// Device/Application/workflowCore
PROGRAM workflowCore
VAR 
	right2All:BOOL;//右扫切全扫标志
	left2All:BOOL;//左扫切全扫标志
	all2Right:BOOL;//全扫切右扫标志
	all2Left:BOOL;//全扫切左扫标志
	leftSweeperSwingOutTemp:BOOL;//左扫摆出中间变量
	rightSweeperSwingOutTemp:BOOL;//右扫摆出中间变量
	ton1:TON;//左扫盘延时下放定时器
	ton2:TON;//左扫盘下放控制延时定时器
	ton3:TON;//右扫盘延时下放定时器
	ton4:TON;//右扫盘下放控制延时定时器
	ton5:TON;//吸嘴延时下降定时器
	ton6:TON;//吸嘴下降持续时间定时器
	ton7:TON;//左扫延时旋转定时器
	ton8:TON;//右扫延时旋转定时器
	ton9:TON;//全扫延时旋转定时器
	ton10:TON;//右扫切全扫定时器
	ton11:TON;//左扫切全扫定时器
	ton12:TON;//全扫切右扫定时器
	ton13:TON;//全扫切左扫定时器
	ton14:TON;//左扫盘上升定时器
	ton15:TON;//右扫盘上升定时器
	ton16:TON;//吸嘴上升定时器
	ton17:TON;//中喷杆球阀定时器
	ton18:TON;//左喷杆球阀定时器
	ton19:TON;//右喷杆球阀定时器
	ton20:TON;//喷雾降尘泵定时器
	tof1:TOF;//左扫盘延时回收定时器
	tof2:TOF;//右扫盘延时回收定时器
	rTrigger1:R_TRIG;//全洗扫上升沿触发
	rTrigger2:R_TRIG;//左洗扫上升沿触发
	rTrigger3:R_TRIG;//右洗扫上升沿触发
	rTrigger4:R_TRIG;//全扫路上升沿触发
	rTrigger5:R_TRIG;//左扫路上升沿触发
	rTrigger6:R_TRIG;//右扫路上升沿触发
	rTrigger7:R_TRIG;//系统工作状态上升沿触发
	
	fTrigger1:F_TRIG;//左扫盘旋转下降沿触发
	fTrigger2:F_TRIG;//右扫盘旋转下降沿触发
	fTrigger3:F_TRIG;//全扫盘旋转下降沿触发	
	fTrigger4:F_TRIG;//系统工作状态下降沿触发
END_VAR

rTrigger1(CLK:= systemStatus.allWashSweep);//全洗扫上升沿触发
rTrigger2(CLK:= systemStatus.leftWashSweep);//左洗扫上升沿触发
rTrigger3(CLK:= systemStatus.rightWashSweep);//右洗扫上升沿触发
rTrigger4(CLK:= systemStatus.allSweep);//全扫路上升沿触发
rTrigger5(CLK:= systemStatus.leftSweep);//左扫路上升沿触发
rTrigger6(CLK:= systemStatus.rightSweep);//右扫路上升沿触发


leftSweeperSwingOutTemp := (systemStatus.allWashSweep OR systemStatus.leftWashSweep OR systemStatus.allSweep OR systemStatus.leftSweep); //左扫摆出中间变量
//左扫即时摆出，延时3S回收
tof1(IN:=leftSweeperSwingOutTemp,PT:=T#3S);
systemStatus.leftSweeperSwingOut:=tof1.Q;
//左扫延时5S下放，控制下放气阀5S得电后失电（保持下放状态）
ton1(IN:=leftSweeperSwingOutTemp,PT:=T#5S);
ton2(IN:=ton1.Q,PT:=T#5S);
systemStatus.leftSweeperDown:=ton1.Q AND (NOT ton2.Q);

rightSweeperSwingOutTemp := (systemStatus.allWashSweep OR systemStatus.rightWashSweep OR systemStatus.allSweep OR systemStatus.rightSweep); //右扫摆出中间变量
//右扫即时摆出，延时3S回收
tof2(IN:=rightSweeperSwingOutTemp,PT:=T#5S);
systemStatus.rightSweeperSwingOut:=tof2.Q;
//右扫延时5S下放，控制下放气阀5S得电后失电（保持下放状态）
ton3(IN:=rightSweeperSwingOutTemp,PT:=T#5S);
ton4(IN:=ton3.Q,PT:=T#5S);
systemStatus.rightSweeperDown:=ton3.Q AND (NOT ton4.Q);

//吸嘴在7S后下降，然后下降过程持续7S
ton5(IN:=systemStatus.systemWork,PT:=T#7S);
ton6(IN:=ton5.Q,PT:=T#7S);
systemStatus.suctionNozzleDown:=ton5.Q AND (NOT ton6.Q);

//左扫盘在12S后旋转
ton7(IN:= systemStatus.leftWashSweep OR systemStatus.leftSweep,PT:= T#12S);
fTrigger1(CLK:= ton7.Q);
//右扫盘在12S后旋转
ton8(IN:= systemStatus.rightWashSweep OR systemStatus.rightSweep,PT:= T#12S);
fTrigger2(CLK:= ton8.Q);
//左右扫盘在12S后旋转
ton9(IN:= systemStatus.allWashSweep OR systemStatus.allSweep,PT:= T#12S);
fTrigger3(CLK:=ton9.Q);
//左右扫盘旋转标志
systemStatus.allSweeperRotate:= ton9.Q AND (NOT systemStatus.leftSweeperRotate) AND (NOT systemStatus.rightSweeperRotate);
//右扫切全扫
right2All:= ((fTrigger2.Q AND (rTrigger1.Q OR rTrigger4.Q)) OR right2All) AND (NOT systemStatus.leftWashSweep) AND (NOT systemStatus.leftSweep)
AND (NOT systemStatus.allWash) AND (NOT systemStatus.leftWash) AND (NOT systemStatus.rightWash) AND (NOT systemStatus.stopWash) AND (NOT ton10.Q);
ton10(IN:= right2All AND (NOT rTrigger3.Q ) AND (NOT rTrigger6.Q),PT:=T#12S); //右扫切全扫状态持续12S,如果在切换状态中重新切换回右扫保证持续旋转12S

//左扫切全扫
left2All:=((fTrigger1.Q AND (rTrigger1.Q OR rTrigger4.Q)) OR left2All) AND (NOT systemStatus.rightWashSweep) AND (NOT systemStatus.rightSweep)
AND (NOT systemStatus.allWash) AND (NOT systemStatus.leftWash) AND (NOT systemStatus.rightWash) AND (NOT systemStatus.stopWash) AND (NOT ton11.Q);
ton11(IN:= left2All AND (NOT rTrigger2.Q ) AND (NOT rTrigger5.Q),PT:=T#12S); //左扫切全扫状态持续12S,如果在切换状态中重新切换回左扫保证持续旋转12S

//全扫切右扫,存在左扫盘持续旋转12S问题以后考虑完善
all2Right :=((fTrigger3.Q AND (rTrigger3.Q OR rTrigger6.Q)) OR all2Right) AND (NOT systemStatus.leftWashSweep) AND (NOT systemStatus.leftSweep)
AND (NOT systemStatus.allWash) AND (NOT systemStatus.leftWash) AND (NOT systemStatus.rightWash) AND (NOT systemStatus.stopWash) AND (NOT ton12.Q);
ton12(IN:= all2Right AND (NOT rTrigger1.Q ) AND (NOT rTrigger4.Q),PT:=T#12S); //全扫切右扫状态持续12S,如果在切换状态中重新切换回全扫保证持续旋转12S

//全扫切左扫,存在右扫盘持续旋转12S问题以后考虑完善
all2Left :=((fTrigger3.Q AND (rTrigger2.Q OR rTrigger5.Q)) OR all2Left) AND (NOT systemStatus.rightWashSweep) AND (NOT systemStatus.rightSweep)
AND (NOT systemStatus.allWash) AND (NOT systemStatus.leftWash) AND (NOT systemStatus.rightWash) AND (NOT systemStatus.stopWash) AND (NOT ton13.Q);
ton13(IN:= all2Left AND (NOT rTrigger1.Q ) AND (NOT rTrigger4.Q),PT:=T#12S); //全扫切左扫状态持续12S,如果在切换状态中重新切换回全扫保证持续旋转12S

//左扫盘旋转标志
systemStatus.leftSweeperRotate:= (ton7.Q OR left2All OR all2Left) AND (NOT systemStatus.allSweeperRotate) AND (NOT systemStatus.rightSweeperRotate);

//右扫盘旋转标志
systemStatus.rightSweeperRotate:= (ton8.Q OR right2All OR all2Right) AND (NOT systemStatus.allSweeperRotate) AND (NOT systemStatus.leftSweeperRotate);

//右洗扫、右扫路、全清洗、左清洗、右清洗、停扫，左扫盘上升，上升气阀得电5S后失电（保持上升状态）
ton14(IN:= systemStatus.rightWashSweep OR systemStatus.rightSweep OR systemStatus.stopWash OR systemStatus.allWash OR systemStatus.leftWash 
OR systemStatus.rightWash,PT:=T#5S);
systemStatus.leftSweeperUp := (systemStatus.rightWashSweep OR systemStatus.rightSweep OR systemStatus.stopWash OR systemStatus.allWash
 OR systemStatus.leftWash OR systemStatus.rightWash) AND (NOT ton14.Q);

//左洗扫、左扫路、全清洗、左清洗、右清洗、停扫，右扫盘上升，上升气阀得电5S后失电（保持上升状态）
ton15(IN:= systemStatus.leftWashSweep OR systemStatus.leftSweep OR systemStatus.stopWash OR systemStatus.allWash OR systemStatus.leftWash 
OR systemStatus.rightWash,PT:=T#5S);
systemStatus.rightSweeperUp:= (systemStatus.leftWashSweep OR systemStatus.leftSweep OR systemStatus.stopWash OR systemStatus.allWash 
OR systemStatus.leftWash OR systemStatus.rightWash) AND (NOT ton15.Q);

//停机，吸嘴上升，即时上升，上升过程持续7S
ton16(IN:=systemStatus.stopWash,PT:=T#7S);
systemStatus.suctionNozzleUp:= systemStatus.stopWash AND (NOT ton16.Q);

//全洗扫、左洗扫、右洗扫、全清洗、左清洗、右清洗，系统在7s后打开中喷杆球阀，开始喷水
ton17(IN:=systemStatus.allWashSweep OR systemStatus.leftWashSweep OR systemStatus.rightWashSweep OR systemStatus.allWash OR systemStatus.leftWash OR systemStatus.rightWash,PT:=T#7S);
systemStatus.centreSprayRodOpen1:= ton17.Q;

//全洗扫、右洗扫、全清洗、右清洗，系统在7S后左喷杆摆出,并左喷杆球阀打开开始喷水
ton18(IN:= systemStatus.allWashSweep OR systemStatus.leftWashSweep OR systemStatus.allWash OR systemStatus.leftWash,PT:= T#7S);
systemStatus.leftSprayRodOpen1:= ton18.Q;//左喷杆球阀打开喷水
systemStatus.leftSprayRodSwingOut:= ton18.Q ;//左喷杆摆出

//全洗扫、右洗扫、全清洗、右清洗，系统在7S后右喷杆摆出,并右喷杆球阀打开开始喷水
ton19(IN:= systemStatus.allWashSweep OR systemStatus.rightWashSweep OR systemStatus.allWash OR systemStatus.rightWash,PT:=T#7S);
systemStatus.rightSprayRodOpen1:= ton19.Q;//右喷杆球阀打开喷水
systemStatus.rightSprayRodSwingOut:= ton19.Q ;//右喷杆摆出

//洗扫和扫路模式触发，设置扫盘配置转速
IF (rTrigger1.Q OR rTrigger2.Q OR rTrigger3.Q OR rTrigger4.Q OR rTrigger5.Q OR rTrigger6.Q)THEN
	//设置为扫盘高速
	IF systemConfig.dspSweeperSpeed = 0 THEN
		systemStatus.sweeperSpeedLow:=FALSE;
		systemStatus.sweeperSpeedMiddle:=FALSE;
		systemStatus.sweeperSpeedHigh:=TRUE;
	END_IF
	//设置为扫盘中速
	IF systemConfig.dspSweeperSpeed =1 THEN
		systemStatus.sweeperSpeedLow:=FALSE;
		systemStatus.sweeperSpeedMiddle:=TRUE;
		systemStatus.sweeperSpeedHigh:=FALSE;
	END_IF
	//设置为扫盘低速
	IF systemConfig.dspSweeperSpeed =2 THEN
		systemStatus.sweeperSpeedLow:=TRUE;
		systemStatus.sweeperSpeedMiddle:=FALSE;
		systemStatus.sweeperSpeedHigh:=FALSE;
	END_IF
END_IF

//扫路模式下，系统在7S后启动喷雾降尘泵
//ton20(IN:= systemStatus.allSweep OR systemStatus.leftSweep OR systemStatus.rightSweep,PT:=T#7S);
//systemStatus.diaphragmPumpStart:= systemConfig.dspDiaphragmPump AND ton20.Q AND input40A.mainWateraValve AND (NOT faultSt.frontTankWaterLevelLow) AND (NOT  faultST.backTankWaterLevelLow);


//扫路模式下，系统启动后断开水泵离合器,进一步考虑降低发动机转速后再分离
IF (rTrigger4.Q OR rTrigger5.Q OR rTrigger6.Q) THEN
	systemStatus.waterPumpConnect:= FALSE;
END_IF

//系统工作，调节发动机转速
rTrigger7(CLK:=systemStatus.systemWork);//系统工作状态上升沿触发
fTrigger4(CLK:=systemStatus.systemWork);//系统工作状态下降沿触发
IF rTrigger7.Q THEN
	systemStatus.engineSetSpeed:= systemConfig.dspEngineStandardSpeed;//调节到标准速度
END_IF
IF fTrigger4.Q AND (NOT systemStatus.AIModel) THEN
	systemStatus.engineSetSpeed:= systemConfig.dspEngineIdlingSpeed;//调节到怠速
	
END_IF

END_PROGRAM

// Device/Application/workflowOther
PROGRAM workflowOther
VAR
	waterPumpWorkCondition :BOOL; //水泵啮合限定条件
	initFlag:BOOL:=0;//程序初始化标志
	
	rTrigger1:R_TRIG;//左角冲_屏输入上升沿触发
	rTrigger2:R_TRIG;//右角冲_屏输入上升沿触发
	rTrigger3:R_TRIG;//后喷雾_屏输入上升沿触发
	rTrigger4:R_TRIG;//手持喷枪_屏输入上升沿触发
	rTrigger5:R_TRIG;//自洁_屏输入上升沿触发
	rTrigger6:R_TRIG;//左前冲_屏输入上升沿触发
	rTrigger7:R_TRIG;//右前冲_屏输入上升沿触发
	rTrigger8:R_TRIG;//左后洒_屏输入上升沿触发
	rTrigger9:R_TRIG;//右后洒_屏输入上升沿触发
	rTrigger10:R_TRIG;//扫盘低速_屏输入上升沿触发
	rTrigger11:R_TRIG;//扫盘中速_屏输入上升沿触发
	rTrigger12:R_TRIG;//扫盘高速_屏输入上升沿触发
	rTrigger13:R_TRIG;//垃圾箱门关_屏输入上升沿触发
	rTrigger14:R_TRIG;//垃圾箱门开_屏输入上升沿触发
	rTrigger15:R_TRIG;//垃圾箱体降_屏输入上升沿触发
	rTrigger16:R_TRIG;//垃圾箱体升_屏输入上升沿触发
	rTrigger17:R_TRIG;//扫刷更换_屏输入上升沿触发
	rTrigger18:R_TRIG;//自动排水_屏输入上升沿触发
	rTrigger19:R_TRIG;//手动排水_屏输入上升沿触发
	rTrigger20:R_TRIG;//智能洗扫_屏输入上升沿触发
	rTrigger21:R_TRIG;//系统工作状态上升沿触发
	rTrigger22:R_TRIG;//车速<8km/h上升沿触发
	rTrigger23:R_TRIG;//车速>8km/h<12km/h上升沿触发
	rTrigger24:R_TRIG;//车速>12km/h<16km/h上升沿触发
	rTrigger25:R_TRIG;//车速大于16km/h上升沿触发
	rTrigger26:R_TRIG;	//转速增加_屏输入上升沿触发
	rTrigger27:R_TRIG;	//转速降低_屏输入上升沿触发
	rTrigger28:R_TRIG;	//标准速度_屏输入上升沿触发
	rTrigger29:R_TRIG;	//强力速度_屏输入上升沿触发
	rTrigger30:R_TRIG;  //工作灯_屏输入上升沿触发
	rTrigger31:R_TRIG;  //隔膜泵_屏输入上升沿触发
	rTrigger32:R_TRIG;  //水泵离合器_屏输入上升沿触发
	rTrigger33:R_TRIG;  //水泵离合器_配置上升沿触发
	
	
	
	tp1:TP;//高压水泵未啮合保持定时器1
	tp2:TP;//总水阀未打开保持定时器1
	tp3:TP;//吹净球阀未关闭保持定时器
	tp4:TP;//箱门未打开保持定时器
	tp5:TP;//左支撑杆未放下保持定时器
	tp6:TP;//右支撑杆未放下保持定时器
	tp7:TP;//发动机未关闭保持定时器
	tp8:TP;//总水阀未打开保持定时器2
	tp9:TP;//吹净球阀未关闭保持定时器2
	
	ton1:TON;//左喷杆排水定时器
	ton2:TON;//右喷杆排水定时器
	ton3:TON;//中喷杆排水定时器
	ton4:TON;//辅助排水定时器
	ton5:TON;//自洁排水定时器
	ton6:ton;//状态1定时器
	ton7:ton;//状态2定时器
	ton8:ton;//状态3定时器
	ton9:ton;//状态4定时器
	ton10:ton;//状态5定时器
	counter:INT;//循环次数
	
	
	fTrigger1:F_TRIG;//高压水泵啮合下降沿触发
	fTrigger2:F_TRIG;//系统工作状态下降沿触发
	fTrigger3:F_TRIG;//发动机工作状态下降沿触发
	fTrigger4:F_TRIG; //水泵离合器_配置下降沿触发
	vehicleSpeed:WORD;//车速
	
END_VAR

//高压水泵啮合限定条件，发动机未工作，吹净球阀关闭，总水阀打开，没有水路卸荷阀未打开故障,没有缺水故障，没有超速故障
 waterPumpWorkCondition:= (NOT systemStatus.engineWork) AND input40A.cleanValve AND input40A.mainWateraValve AND (NOT faultST.waterUnloadValveNotOpen)
	   AND (NOT faultST.frontTankWaterLevelLow) AND (NOT faultST.backTankWaterLevelLow) AND (NOT faultST.highPressurePumpOverSpeedStop);
//程序重启时配置生效
IF NOT initFlag THEN
	systemStatus.waterPumpConnect:=systemConfig.dspWaterPumpConnect AND waterPumpWorkCondition;//导入配置
	initFlag:=TRUE;
END_IF	
//  程序运行时配置即时生效 
rTrigger33(clk:=systemConfig.dspWaterPumpConnect);
fTrigger4(clk:=systemConfig.dspWaterPumpConnect);
IF  rTrigger33.Q OR fTrigger4.Q THEN
	systemStatus.waterPumpConnect:=systemConfig.dspWaterPumpConnect AND waterPumpWorkCondition;//配置即时生效
END_IF
//水泵离合器啮合操作（水泵离合器必须静止啮合）
rTrigger32(clk:=dspSystemInput.dspWaterPumpDisconnect);
IF rTrigger32.Q THEN
	IF systemStatus.waterPumpConnect THEN
		systemStatus.waterPumpConnect:=FALSE;
	ELSE
		systemStatus.waterPumpConnect:=waterPumpWorkCondition;
	END_IF
END_IF
//提示信息
//发动机未关闭
tp7(IN:=rTrigger32.Q AND NOT systemStatus.engineWork,PT:=T#1S);
tipsST.stopEngineFirst:= tp7.Q;
//总水阀未打开
tp8(IN:= rTrigger32.Q AND (NOT input40A.mainWateraValve),PT:=T#1S);
tipsST.mainWateraValveNotOpen4:= tp8.Q;  //总水阀未打开判断
//吹净球阀未关闭
tp9(IN:= rTrigger32.Q AND (NOT input40A.cleanValve),PT:=T#1S);     
tipsST.cleanValveNotClose4:= tp9.Q;       //在吹净球阀未关闭判断  
//如果水泵啮合后出现故障，将自动断开
IF systemStatus.waterPumpConnect THEN
	systemStatus.waterPumpConnect:= input40A.cleanValve AND input40A.mainWateraValve AND (NOT faultST.waterUnloadValveNotOpen)
	   AND (NOT faultST.frontTankWaterLevelLow) AND (NOT faultST.backTankWaterLevelLow) AND (NOT faultST.highPressurePumpOverSpeedStop);
END_IF

fTrigger1(CLK:=systemStatus.waterPumpConnect);//高压水泵啮合下降沿触发
//左角冲
rTrigger1(CLK:=dspSystemInput.dspLeftFlush);
IF (rTrigger1.Q AND systemStatus.waterPumpConnect) THEN
	IF systemStatus.leftFlushOpen THEN
		systemStatus.leftFlushOpen:=FALSE;
		IF (NOT systemStatus.sprayGun) AND (NOT systemStatus.backSprayOpen) AND (NOT systemStatus.rightFlushOpen) THEN
			systemStatus.auxiliaryValveOpen1:=FALSE;
			systemStatus.engineSetSpeed:=systemConfig.dspEngineIdlingSpeed;//调节发动机转速到怠速
		END_IF
	ELSE
		systemStatus.leftFlushOpen:=systemStatus.waterPumpConnect;
		IF systemStatus.leftFlushOpen THEN
		systemStatus.auxiliaryValveOpen1:=TRUE;
        systemStatus.engineSetSpeed:=1200;//调节发动机转速,???
	   END_IF
	END_IF	
END_IF
IF fTrigger1.Q THEN
	systemStatus.leftFlushOpen:=FALSE;
END_IF
//右角冲
rTrigger2(CLK:=dspSystemInput.dspRightFlush);
IF rTrigger2.Q THEN
	IF systemStatus.rightFlushOpen THEN
		systemStatus.rightFlushOpen:=FALSE;
		IF (NOT systemStatus.sprayGun) AND (NOT systemStatus.backSprayOpen) AND (NOT systemStatus.leftFlushOpen) THEN
			systemStatus.auxiliaryValveOpen1:=FALSE;
			systemStatus.engineSetSpeed:=systemConfig.dspEngineIdlingSpeed;//调节发动机转速到怠速
		END_IF	
	ELSE
		systemStatus.rightFlushOpen:=systemStatus.waterPumpConnect;	
        IF systemStatus.rightFlushOpen THEN
		    systemStatus.auxiliaryValveOpen1:=TRUE;
		    systemStatus.engineSetSpeed:=1200;//调节发动机转速,???
	    END_IF
	END_IF	
END_IF
IF fTrigger1.Q THEN
	systemStatus.rightFlushOpen:=FALSE;
END_IF
//后喷雾
rTrigger3(CLK:=dspSystemInput.dspBackSpray);
IF rTrigger3.Q THEN
	IF systemStatus.backSprayOpen THEN
		systemStatus.backSprayOpen:=FALSE;
		IF (NOT systemStatus.sprayGun) AND (NOT systemStatus.rightFlushOpen) AND (NOT systemStatus.leftFlushOpen) THEN
			systemStatus.auxiliaryValveOpen1:=FALSE;
			systemStatus.engineSetSpeed:=systemConfig.dspEngineIdlingSpeed;//调节发动机转速到怠速
		END_IF	
	ELSE
		systemStatus.backSprayOpen:=systemStatus.waterPumpConnect;
		IF systemStatus.backSprayOpen THEN
			systemStatus.auxiliaryValveOpen1:=TRUE;
		    systemStatus.engineSetSpeed:=1200;//调节发动机转速,???
	    END_IF
	END_IF
END_IF
IF fTrigger1.Q THEN
	systemStatus.backSprayOpen:=FALSE;
END_IF
//手持喷枪
rTrigger4(CLK:=dspSystemInput.dspSprayGun);
IF rTrigger4.Q THEN
	IF systemStatus.sprayGun THEN
		systemStatus.sprayGun:=FALSE;
		IF (NOT systemStatus.backSprayOpen) AND (NOT systemStatus.rightFlushOpen) AND (NOT systemStatus.leftFlushOpen) THEN
			systemStatus.auxiliaryValveOpen1:=FALSE;
			systemStatus.engineSetSpeed:=systemConfig.dspEngineIdlingSpeed;//调节发动机转速到怠速
		END_IF		
	ELSE
		systemStatus.sprayGun:=systemStatus.waterPumpConnect;
		IF systemStatus.sprayGun THEN
			systemStatus.auxiliaryValveOpen1:=TRUE;
		    systemStatus.engineSetSpeed:=1200;//调节发动机转速,???
	    END_IF
	END_IF	
	panelInput.sprayGunFlag:=systemStatus.sprayGun;//触摸屏和硅胶面板两点控制
END_IF
IF fTrigger1.Q THEN
	systemStatus.sprayGun:=FALSE;
END_IF
//自洁
rTrigger5(CLK:=dspSystemInput.dspSelfClean);
IF rTrigger5.Q THEN
	IF systemStatus.selfClean THEN
		systemStatus.selfClean:=FALSE;
		
	ELSE			
        systemStatus.selfClean:=systemStatus.waterPumpConnect;
		IF systemStatus.selfClean THEN
		  systemStatus.selfSprayRodOpen1:=TRUE;
		  systemStatus.engineSetSpeed:=1200;//调节发动机转速,???
	    END_IF
	END_IF	
	panelInput.selfCleanFlag:=systemStatus.selfClean; //硅胶面板和触摸屏两点自洁控制
END_IF
IF fTrigger1.Q THEN
	systemStatus.selfClean:=FALSE;
END_IF
//提示信息
//高压水泵未啮合
tp1(IN:=(rTrigger1.Q AND (NOT systemStatus.leftFlushOpen) AND (NOT systemStatus.waterPumpConnect)) OR
                   (rTrigger2.Q AND (NOT systemStatus.rightFlushOpen) AND (NOT systemStatus.waterPumpConnect)) OR
				   (rTrigger3.Q AND (NOT systemStatus.backSprayOpen) AND (NOT systemStatus.waterPumpConnect)) OR
				   (rTrigger4.Q AND (NOT systemStatus.sprayGun) AND (NOT systemStatus.waterPumpConnect)) OR
				   (rTrigger5.Q AND (NOT systemStatus.selfClean) AND (NOT systemStatus.waterPumpConnect)),PT:=T#2S) ;
tipsST.highPressurePumpDisconnect3:=	tp1.Q;//高压水泵未啮合判断
//总水阀未打开
//tp2(IN:= tipsST.highPressurePumpDisconnect3 AND (NOT input40A.mainWateraValve),PT:=T#1S);
//tipsST.mainWateraValveNotOpen3:= tp2.Q;  //在workflowCore()存在高总水阀未打开判断
//吹净球阀未关闭
//tp3(IN:= tipsST.highPressurePumpDisconnect3 AND (NOT input40A.cleanValve),PT:=T#1S);     
//tipsST.cleanValveNotClose3:= tp3.Q ;       //在workflowCore()存在吹净球阀未关闭判断   

//左前冲洗
rTrigger6(CLK:=dspSystemInput.dspLeftFrontSprinkle);
IF (rTrigger6.Q AND (NOT systemStatus.systemTest)) THEN
	systemStatus.leftFrontSprinkle:= NOT systemStatus.leftFrontSprinkle;
END_IF

//右前冲洗
rTrigger7(CLK:=dspSystemInput.dspRightFrontSprinkle);
IF (rTrigger7.Q AND (NOT systemStatus.systemTest)) THEN
	systemStatus.rightFrontSprinkle:= NOT systemStatus.rightFrontSprinkle;
END_IF

//左后洒
rTrigger8(CLK:=dspSystemInput.dspLeftBackSprinkle);
IF (rTrigger8.Q AND (NOT systemStatus.systemTest)) THEN
	systemStatus.leftBackSprinkle:=NOT systemStatus.leftBackSprinkle;
END_IF

//右后洒
rTrigger9(CLK:=dspSystemInput.dspRightBackSprinkle);
IF (rTrigger9.Q AND (NOT systemStatus.systemTest)) THEN
	systemStatus.rightBackSprinkle:=NOT systemStatus.rightBackSprinkle;
END_IF

//扫盘低速
rTrigger10(CLK:=dspSystemInput.dspSweeperSpeedLow);
IF rTrigger10.Q THEN
		systemStatus.sweeperSpeedLow:=TRUE;
		systemStatus.sweeperSpeedMiddle:=FALSE;
		systemStatus.sweeperSpeedHigh:=FALSE;
END_IF

//扫盘中速
rTrigger11(CLK:=dspSystemInput.dspSweeperSpeedMiddle);
IF rTrigger11.Q THEN
		systemStatus.sweeperSpeedLow:=FALSE;
		systemStatus.sweeperSpeedMiddle:=TRUE;
		systemStatus.sweeperSpeedHigh:=FALSE;
END_IF

//扫盘高速
rTrigger12(CLK:=dspSystemInput.dspSweeperSpeedHigh);
IF rTrigger12.Q THEN
		systemStatus.sweeperSpeedLow:=FALSE;
		systemStatus.sweeperSpeedMiddle:=FALSE;
		systemStatus.sweeperSpeedHigh:=TRUE;
END_IF

//箱门关
systemStatus.tankDoorClose:= dspSystemInput.dspTankDoorClose AND (NOT dspSystemInput.dspTankDoorOpen) AND (NOT systemStatus.tankDoorOpen) AND (NOT panelInput.tankDoorOpenFlag);

//箱门开
systemStatus.tankDoorOpen:= dspSystemInput.dspTankDoorOpen AND (NOT dspSystemInput.dspTankDoorClose) AND (NOT systemStatus.tankDoorClose) AND (NOT panelInput.tankDoorCloseFlag) ;
	
//箱体升
systemStatus.tankUp:= dspSystemInput.dspTankUp AND (NOT dspSystemInput.dspTankDown ) AND (NOT input40A.backDoor) AND (NOT systemStatus.tankDown) AND (NOT panelInput.tankDownFlag);

//箱体降
systemStatus.tankDown:= dspSystemInput.dspTankDown AND (NOT dspSystemInput.dspTankUp ) AND  input40A.leftRod AND input40A.rightRod AND (NOT systemStatus.tankUp) AND (NOT panelInput.tankUpFlag);

//提示
//箱门未打开
tp4(IN:= (dspSystemInput.dspTankUp AND input40A.backDoor),PT:=T#1S);
tipsST.tankDoorNotOpen:=tp4.Q;
//左支撑杆未放下
tp5(IN:=dspSystemInput.dspTankDown AND NOT input40A.leftRod,PT:=T#1S);
tipsST.leftRodUp:=tp5.Q;
//右支撑杆未放下
tp6(IN:=dspSystemInput.dspTankDown AND NOT input40A.rightRod,PT:=T#1S);
tipsST.rightRodUp:=tp6.Q;

//扫刷更换
rTrigger17(CLK:= dspSystemInput.dspReplaceSweeper);
IF rTrigger17.Q AND (NOT systemStatus.engineWork) THEN
	systemStatus.replaceSweeper:=NOT systemStatus.replaceSweeper;
END_IF
IF dspSystemInput.dspEngineStart THEN
	systemStatus.replaceSweeper:=FALSE;
END_IF

//工作灯,触摸屏和硅胶面板皆可控制
rTrigger30(CLK:=dspSystemInput.dspWorkLamp);
IF rTrigger30.Q THEN
	systemStatus.workLamp:=NOT systemStatus.workLamp;
	panelInput.workLampFlag:=systemStatus.workLamp;
END_IF

//隔膜泵
rTrigger31(CLK:=dspSystemInput.dspDiaphragmPump);
IF rTrigger31.Q THEN
	IF systemStatus.diaphragmPump THEN
		systemStatus.diaphragmPump:=FALSE;
	ELSE
		systemStatus.diaphragmPump:=input40A.mainWateraValve AND (NOT faultST.frontTankWaterLevelLow) AND (NOT  faultST.backTankWaterLevelLow);
	END_IF
END_IF

//排水控制
//自动和手动切换控制
rTrigger18(CLK:=dspSystemInput.dspAutoDrainOff);//自动排水_屏输入上升沿触发
rTrigger19(CLK:=dspSystemInput.dspManualDrainOff);//手动排水_屏输入上升沿触发
IF rTrigger18.Q THEN
	IF systemStatus.autoDrainOff THEN
		systemStatus.autoDrainOff:=FALSE;
	ELSE
		systemStatus.autoDrainOff:= NOT systemStatus.engineWork;
        IF systemStatus.autoDrainOff THEN
			counter:=3;//自动循环次数
		    systemStatus.manualDrainOff:= FALSE;
	    END_IF	
	END_IF	
END_IF
IF rTrigger19.Q AND (NOT systemStatus.engineWork) THEN
	systemStatus.manualDrainOff:=TRUE;
	systemStatus.autoDrainOff:= FALSE;	
END_IF
IF dspSystemInput.dspEngineStart THEN
	systemStatus.manualDrainOff:=FALSE;
	systemStatus.autoDrainOff:= FALSE;	
END_IF
//手动模式
IF systemStatus.manualDrainOff THEN
	systemStatus.auxiliaryValveOpen2:=dspSystemInput.dspAuxiliarySystemDrainOff; //辅助球阀喷水标志
	systemStatus.leftSprayRodOpen2:=dspSystemInput.dspLeftSprayRodDrainOff; //左侧喷杆喷水标志
	systemStatus.selfSprayRodOpen2:=dspSystemInput.dspSelfCleanDrainOff; //自洁喷杆喷水标志
	systemStatus.rightSprayRodOpen2 :=dspSystemInput.dspRightSprayRodDrainOff; //右侧喷杆喷水标志
	systemStatus.centreSprayRodOpen2 :=dspSystemInput.dspCentreSprayRodDrainOff; //中喷杆喷水标志
END_IF
//自动模式
ACT();
//自动模式,循环3次
(*ton1(IN:=systemStatus.autoDrainOff,PT:=T#4S);//左喷杆排水定时器
ton2(IN:=systemStatus.autoDrainOff,PT:=T#8S);//右喷杆排水定时器
ton3(IN:=systemStatus.autoDrainOff,PT:=T#12S);//中喷杆排水定时器
ton4(IN:=systemStatus.autoDrainOff,PT:=T#16S);//辅助排水定时器
ton5(IN:=systemStatus.autoDrainOff,PT:=T#20S);//自洁排水定时器
IF systemStatus.autoDrainOff THEN
	systemStatus.leftSprayRodOpen:=NOT ton1.Q OR systemStatus.leftSprayRodOpen;//左喷杆排水,执行0-4S
    systemStatus.rightSprayRodOpen:= ton1.Q AND (NOT ton2.Q) OR systemStatus.rightSprayRodOpen;//右喷杆排水,4-8s;
	systemStatus.centreSprayRodOpen:=ton2.Q AND (NOT ton3.Q ) OR systemStatus.centreSprayRodOpen;//中喷杆排水，8-12S;
	systemStatus.auxiliaryValveOpen:=ton3.Q AND (NOT ton4.Q ) OR systemStatus.auxiliaryValveOpen;//辅助排水，12-16S;
	systemStatus.selfSprayRodOpen:= ton4.Q AND (NOT ton5.Q ) OR systemStatus.selfSprayRodOpen;//自洁排水，16-20S;
END_IF*)

//智能洗扫模式
rTrigger20(CLK:=dspSystemInput.dspAIModel);//智能洗扫_屏输入上升沿触发
rTrigger21(CLK:=systemStatus.systemWork);//系统工作状态上升沿触发
fTrigger2(CLK:=systemStatus.systemWork);//系统工作状态下降沿触发
fTrigger3(CLK:=systemStatus.engineWork);//发动机工作状态下降沿触发
//按钮控制智能模式
IF rTrigger20.Q THEN
   systemStatus.AIModel:=NOT systemStatus.AIModel;
END_IF
//系统工作配置智能模式
IF rTrigger21.Q THEN
	systemStatus.AIModel:= systemConfig.dspAIModel;
END_IF
IF fTrigger2.Q THEN
	systemStatus.AIModel:=FALSE;
END_IF
IF fTrigger3.Q THEN
	systemStatus.AIModel:=FALSE;
END_IF

IF systemStatus.AIModel AND systemStatus.systemWork THEN
	rTrigger22(CLK:=systemStatus.vehicleSpeed<8);//车速<8km/h上升沿触发
	rTrigger23(CLK:=(8<systemStatus.vehicleSpeed AND systemStatus.vehicleSpeed<12));//车速>8km/h<12km/h上升沿触发
	rTrigger24(CLK:=(12<systemStatus.vehicleSpeed AND systemStatus.vehicleSpeed<16));//车速>12km/h<16km/h上升沿触发
	rTrigger25(CLK:=systemStatus.vehicleSpeed>16);//车速大于16km/h上升沿触发
	IF rTrigger22.Q THEN  //车速小于8km/h
		IF dspSystemInput.dspCleanRoad THEN //清洁路面
			systemStatus.engineSetSpeed:=1000;//调节发动机转速,1000rpm
		END_IF
		IF dspSystemInput.dspNormalRoad THEN //一般路面
			systemStatus.engineSetSpeed:=1200;//调节发动机转速,1200rpm
		END_IF
		IF dspSystemInput.dspDirtyRoad THEN //一般路面
			systemStatus.engineSetSpeed:=1350;//调节发动机转速,1350rpm
		END_IF
     END_IF
	IF rTrigger23.Q THEN  //车速>8km/h,并且<12km/h
		IF dspSystemInput.dspCleanRoad THEN //清洁路面
			systemStatus.engineSetSpeed:=1000;//调节发动机转速,1000rpm
		END_IF
		IF dspSystemInput.dspNormalRoad THEN //一般路面
			systemStatus.engineSetSpeed:=1350;//调节发动机转速,1350rpm
		END_IF
		IF dspSystemInput.dspDirtyRoad THEN //一般路面
			systemStatus.engineSetSpeed:=1550;//调节发动机转速,1550rpm
		END_IF
     END_IF
	 IF rTrigger24.Q THEN  //车速>12km/h,并且<16km/h
		IF dspSystemInput.dspCleanRoad THEN //清洁路面
			systemStatus.engineSetSpeed:=1100;//调节发动机转速,1100rpm
		END_IF
		IF dspSystemInput.dspNormalRoad THEN //一般路面
			systemStatus.engineSetSpeed:=1500;//调节发动机转速,1500rpm
		END_IF
		IF dspSystemInput.dspDirtyRoad THEN //一般路面
			systemStatus.engineSetSpeed:=1750;//调节发动机转速,1750rpm
		END_IF
     END_IF
	 IF rTrigger5.Q THEN  //车速>16km/h
		IF dspSystemInput.dspCleanRoad THEN //清洁路面
			systemStatus.engineSetSpeed:=1450;//调节发动机转速,1450rpm
		END_IF
		IF dspSystemInput.dspNormalRoad THEN //一般路面
			systemStatus.engineSetSpeed:=1750;//调节发动机转速,1750rpm
		END_IF
		IF dspSystemInput.dspDirtyRoad THEN //一般路面
			systemStatus.engineSetSpeed:=1750;//调节发动机转速,1750rpm
		END_IF
     END_IF
   
END_IF

//发动机转速调节
rTrigger26(CLK:=dspSystemInput.dspSpeedUp);//转速增加_屏输入上升沿触发
rTrigger27(CLK:=dspSystemInput.dspSpeedDown);//转速降低_屏输入上升沿触发
rTrigger28(CLK:=dspSystemInput.dspStandardSpeed);//标准速度_屏输入上升沿触发
rTrigger29(CLK:=dspSystemInput.dspStrongSpeed);//强力速度_屏输入上升沿触发
//加速
IF rTrigger26.Q  AND (NOT dspSystemInput.dspSpeedDown) AND systemStatus.engineWork THEN
	systemStatus.engineSetSpeed:= systemStatus.engineSetSpeed+systemConfig.dspIncreaseStep;
	IF systemStatus.engineSetSpeed >  systemConfig.dspEngineMaxSpeed THEN
		systemStatus.engineSetSpeed:=systemConfig.dspEngineMaxSpeed;
	END_IF
END_IF
//减速
IF rTrigger27.Q  AND (NOT dspSystemInput.dspSpeedUp) AND systemStatus.engineWork THEN
	systemStatus.engineSetSpeed:= systemStatus.engineSetSpeed+systemConfig.dspIncreaseStep;
	IF systemStatus.engineSetSpeed < systemConfig.dspEngineIdlingSpeed THEN
		systemStatus.engineSetSpeed:= systemConfig.dspEngineIdlingSpeed;
	END_IF
END_IF
//标准速度
IF rTrigger28.Q  AND (NOT dspSystemInput.dspStrongSpeed) AND systemStatus.engineWork THEN
	systemStatus.engineSetSpeed:= systemConfig.dspEngineStandardSpeed;
END_IF
//强力速度
IF rTrigger29.Q  AND (NOT dspSystemInput.dspStandardSpeed) AND systemStatus.engineWork THEN
	systemStatus.engineSetSpeed:= systemConfig.dspEngineStrongSpeed;
END_IF

ACTION ACT:
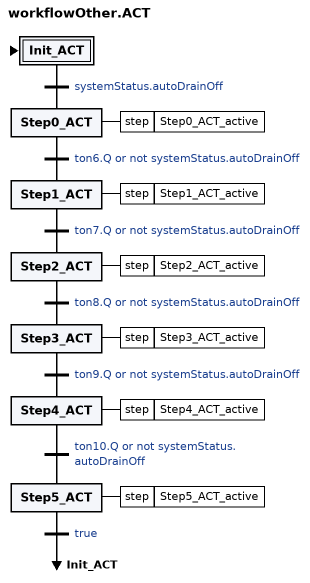
INITIAL_STEP Init_ACT:
END_STEP
TRANSITION FROM Init_ACT TO Step0_ACT
    := systemStatus.autoDrainOff;
END_TRANSITION
STEP Step0_ACT:
    Step0_ACT_active(N);  // step action
END_STEP
TRANSITION FROM Step0_ACT TO Step1_ACT
    := ton6.Q or not systemStatus.autoDrainOff;
END_TRANSITION
STEP Step1_ACT:
    Step1_ACT_active(N);  // step action
END_STEP
TRANSITION FROM Step1_ACT TO Step2_ACT
    := ton7.Q or not systemStatus.autoDrainOff;
END_TRANSITION
STEP Step2_ACT:
    Step2_ACT_active(N);  // step action
END_STEP
TRANSITION FROM Step2_ACT TO Step3_ACT
    := ton8.Q or not systemStatus.autoDrainOff;
END_TRANSITION
STEP Step3_ACT:
    Step3_ACT_active(N);  // step action
END_STEP
TRANSITION FROM Step3_ACT TO Step4_ACT
    := ton9.Q or not systemStatus.autoDrainOff;
END_TRANSITION
STEP Step4_ACT:
    Step4_ACT_active(N);  // step action
END_STEP
TRANSITION FROM Step4_ACT TO Step5_ACT
    := ton10.Q or not systemStatus.autoDrainOff;
END_TRANSITION
STEP Step5_ACT:
    Step5_ACT_active(N);  // step action
END_STEP
TRANSITION FROM Step5_ACT TO Init_ACT
    := true;
END_TRANSITION
END_ACTION

ACTION Step0_ACT_active:
systemStatus.leftSprayRodOpen2:=systemStatus.autoDrainOff AND NOT ton1.Q;
ton1(IN:=TRUE,PT:=T#4S);//左喷杆排水定时器
ton6(IN:=TRUE,PT:=T#10S);//状态1定时器
END_ACTION

ACTION Step1_ACT_active:
systemStatus.leftSprayRodOpen2:=FALSE;
systemStatus.rightSprayRodOpen2:=systemStatus.autoDrainOff AND NOT ton2.Q;
ton2(IN:=TRUE,PT:=T#4S);//右喷杆排水定时器
ton7(IN:=TRUE,PT:=T#10S);//状态2定时器
END_ACTION

ACTION Step2_ACT_active:
systemStatus.rightSprayRodOpen2:=FALSE;
systemStatus.centreSprayRodOpen2:=systemStatus.autoDrainOff AND NOT ton3.Q;
ton3(IN:=TRUE,PT:=T#4S);//中喷杆排水定时器
ton8(IN:=TRUE,PT:=T#10S);//状态3定时器
END_ACTION

ACTION Step3_ACT_active:
systemStatus.centreSprayRodOpen2:=FALSE;
systemStatus.auxiliaryValveOpen2:=systemStatus.autoDrainOff AND ton4.Q;
ton4(IN:=TRUE,PT:=T#4S);//辅助排水定时器
ton9(IN:=TRUE,PT:=T#10S);//状态4定时器
END_ACTION

ACTION Step4_ACT_active:
systemStatus.auxiliaryValveOpen2:=FALSE;
systemStatus.selfSprayRodOpen2:= systemStatus.autoDrainOff AND NOT ton5.Q ;
ton5(IN:=TRUE,PT:=T#4S);//自洁排水定时器
ton10(IN:=TRUE,PT:=T#10S);//状态5定时器
END_ACTION

ACTION Step5_ACT_active:
systemStatus.selfSprayRodOpen2:=FALSE;
counter:=counter-1;
IF counter=0 THEN
	systemStatus.autoDrainOff:=FALSE;
END_IF
//复位定时器
ton1(IN:=FALSE);
ton2(IN:=FALSE);
ton3(IN:=FALSE);
ton4(IN:=FALSE);
ton5(IN:=FALSE);
ton6(IN:=FALSE);
ton7(IN:=FALSE);
ton8(IN:=FALSE);
ton9(IN:=FALSE);
ton10(IN:=FALSE);
END_ACTION

END_PROGRAM

// Device/Application/panelControl
PROGRAM panelControl
VAR
	rTrigger1:R_TRIG;//自洁_硅胶面板上升沿触发
	rTrigger2:R_TRIG;//手持喷枪_硅胶面板上升沿触发
	rTrigger3:R_TRIG;//喷杆伸缩_硅胶面板上升沿触发
	rTrigger4:R_TRIG;//备用动力_硅胶面板上升沿触发
	rTrigger5:R_TRIG;//工作灯_硅胶面板上升沿触发
	rTrigger6:R_TRIG;//背光灯_硅胶面板上升沿触发
	rTrigger7:R_TRIG;//左扫盘下放_硅胶面板上升沿触发
	rTrigger8:R_TRIG;//左扫盘回收_硅胶面板上升沿触发
	rTrigger9:R_TRIG;//右扫盘下放_硅胶面板上升沿触发
	rTrigger10:R_TRIG;//右扫盘回收_硅胶面板上升沿触发
	
	tof1:TOF;//左扫下降延时关断定时器
	tof2:TOF;//右扫下降延时关断定时器
	
	ton1:TON;//左扫下降延时打开定时器1
	ton2:TON;//左扫下降延时打开定时器2
	ton3:TON;//右扫下降延时打开定时器1
	ton4:TON;//右扫下降延时打开定时器2
	
	fTrigger1:F_TRIG;//高压水泵啮合下降沿触发
	
	tp1:TP;//高压水泵未啮合保持定时器
	tp2:TP;//总水阀未打开保持定时器
	tp3:TP;//吹净球阀未关闭保持定时器
END_VAR

//箱门关
panelInput.tankDoorCloseFlag:= panelInput.tankDoorClose AND (NOT panelInput.tankDoorOpen) AND (NOT panelInput.tankDoorOpenFlag);

//箱门开
panelInput.tankDoorOpenFlag:= panelInput.tankDoorOpen  AND (NOT panelInput.tankDoorClose) AND (NOT panelInput.tankDoorCloseFlag) ;
	
//箱体升
panelInput.tankUpFlag:= panelInput.tankUp AND (NOT panelInput.tankDown) AND (NOT panelInput.tankDownFlag);

//箱体降
panelInput.tankDownFlag:= panelInput.tankDown AND (NOT panelInput.tankUp) AND (NOT panelInput.tankUpFlag);

//吸嘴降
panelInput.suctionNozzleDownFlag:= panelInput.suctionNozzleDown AND (NOT systemStatus.systemWork) AND (NOT panelInput.suctionNozzleUp) AND (NOT panelInput.suctionNozzleUpFlag);

//吸嘴升
panelInput.suctionNozzleUpFlag:= panelInput.suctionNozzleUp AND (NOT systemStatus.systemWork) AND (NOT panelInput.suctionNozzleDown) AND (NOT panelInput.suctionNozzleDownFlag);


//自洁
rTrigger1(CLK:=panelInput.selfClean);//自洁_硅胶面板上升沿触发
fTrigger1(CLK:=systemStatus.waterPumpConnect);//高压水泵啮合下降沿触发
IF rTrigger1.Q THEN
	IF panelInput.selfCleanFlag THEN
		panelInput.selfCleanFlag:=FALSE;		
	ELSE			
        panelInput.selfCleanFlag:=systemStatus.waterPumpConnect;
		IF panelInput.selfCleanFlag THEN
		  systemStatus.selfSprayRodOpen1:=TRUE;
		  systemStatus.engineSetSpeed:=1200;//调节发动机转速,???
	    END_IF
	END_IF	
	systemStatus.selfClean:=panelInput.selfCleanFlag;//硅胶面板和触摸屏两点自洁控制
END_IF
IF fTrigger1.Q THEN
	panelInput.selfCleanFlag:=FALSE;
END_IF

//手持喷枪
rTrigger2(CLK:=panelInput.sprayGun);
IF rTrigger2.Q THEN
	IF panelInput.sprayGunFlag THEN
		panelInput.sprayGunFlag:=FALSE;
		IF (NOT systemStatus.backSprayOpen) AND (NOT systemStatus.rightFlushOpen) AND (NOT systemStatus.leftFlushOpen) THEN
			systemStatus.auxiliaryValveOpen1:=FALSE;
			systemStatus.engineSetSpeed:=systemConfig.dspEngineIdlingSpeed;//调节发动机转速到怠速
		END_IF	
	ELSE
		panelInput.sprayGunFlag:=systemStatus.waterPumpConnect;
		IF panelInput.sprayGunFlag THEN
			systemStatus.auxiliaryValveOpen1:=TRUE;
		    systemStatus.engineSetSpeed:=1200;//调节发动机转速,???
	    END_IF
	END_IF	
	systemStatus.sprayGun:=panelInput.sprayGunFlag;//触摸屏和硅胶面板两点控制
END_IF
IF fTrigger1.Q THEN
	panelInput.sprayGunFlag:=FALSE;
END_IF
//提示信息
//高压水泵未啮合
tp1(IN:=(rTrigger1.Q AND (NOT panelInput.selfCleanFlag) AND (NOT systemStatus.waterPumpConnect) OR
         (rTrigger2.Q AND (NOT panelInput.sprayGunFlag) AND (NOT systemStatus.waterPumpConnect))),PT:=T#2S) ;
tipsST.highPressurePumpDisconnect2:=tp1.Q ;//高压水泵未啮合判断
//总水阀未打开
//tp2(IN:= tipsST.highPressurePumpDisconnect2 AND (NOT input40A.mainWateraValve),PT:=T#1S);
//tipsST.mainWateraValveNotOpen2:= tp2.Q;  //高总水阀未打开判断
//吹净球阀未关闭
//tp3(IN:= tipsST.highPressurePumpDisconnect2 AND (NOT input40A.mainWateraValve),PT:=T#1S);     
//tipsST.cleanValveNotClose2:= tp3.Q;       //吹净球阀未关闭判断  

//喷杆伸缩,与测试的喷杆摆出按钮互锁
rTrigger3(CLK:=panelInput.sprayRodOutOrIn);
IF rTrigger3.Q THEN
	IF panelInput.sprayRodOutOrInFlag THEN 
		panelInput.sprayRodOutOrInFlag:=FALSE;
	ELSE
		panelInput.sprayRodOutOrInFlag:=(NOT ctlTestFlag.ctlLeftSprayRodSwingOutTest) AND (NOT ctlTestFlag.ctlRightSprayRodSwingOutTest) AND (NOT systemStatus.systemWork);	
	END_IF
END_IF

//备用动力
//备用动力置位表示在硅胶面板执行吸嘴升降、箱体升降、箱门开闭的时候会随着动作执行而启动，随着动作关闭而延时5秒关闭,并且发动机打开的情况下不会打开备用动力
rTrigger4(CLK:=panelInput.backupMotor);	
IF rTrigger4.Q THEN
	panelInput.backupMotorFlag:= NOT panelInput.backupMotorFlag;
END_IF

systemStatus.backupMotorOpen:= panelInput.suctionNozzleDownFlag OR panelInput.suctionNozzleUpFlag OR panelInput.tankDownFlag OR
                           panelInput.tankUpFlag OR panelInput.tankDoorCloseFlag OR panelInput.tankDoorOpenFlag AND systemStatus.engineWork AND
						   panelInput.backupMotorFlag;

//工作灯,触摸屏和硅胶面板皆可控制
rTrigger5(CLK:=panelInput.workLamp);	
IF rTrigger5.Q THEN
	panelInput.workLampFlag:=NOT panelInput.workLampFlag;
	systemStatus.workLamp:=panelInput.workLampFlag;
END_IF

//背光灯
rTrigger6(CLK:=panelInput.backlight);	
IF rTrigger6.Q THEN
	panelInput.backlightFlag:=NOT panelInput.backlightFlag;
END_IF
 
//左扫盘下放
rTrigger7(CLK:=panelInput.leftSweeperOutAndDown);
IF rTrigger7.Q  THEN
	IF NOT systemStatus.systemWork THEN
		panelInput.leftSweeperOutAndDownFlag:=TRUE;
		panelInput.leftSweeperUpAndInFlag:=FALSE;
	END_IF
END_IF
//左扫盘回收
rTrigger8(CLK:=panelInput.leftSweeperUpAndIn);
IF rTrigger8.Q  THEN
	IF NOT systemStatus.systemWork THEN
		panelInput.leftSweeperOutAndDownFlag:=FALSE;
		panelInput.leftSweeperUpAndInFlag:=TRUE;
	END_IF
END_IF 

//左扫即时摆出，延时3S回收
tof1(IN:=panelInput.leftSweeperOutAndDownFlag,PT:=T#3S);
systemStatus.leftSweeperSwingOut:=tof1.Q AND (NOT systemStatus.systemWork) OR systemStatus.leftSweeperSwingOut;//保证系统工作的情况下，系统工作动作优先
//左扫延时5S下放，控制下放气阀5S得电后失电（保持下放状态）
ton1(IN:=panelInput.leftSweeperOutAndDownFlag,PT:=T#5S);
ton2(IN:=ton1.Q,PT:=T#5S);
systemStatus.leftSweeperDown:=ton1.Q AND (NOT ton2.Q) AND (NOT systemStatus.systemWork) OR systemStatus.leftSweeperDown;//保证系统工作的情况下，系统工作动作优先

//右扫盘下放
rTrigger9(CLK:=panelInput.rightSweeperOutAndDown);
IF rTrigger9.Q  THEN
	IF NOT systemStatus.systemWork THEN
		panelInput.rightSweeperOutAndDownFlag:=TRUE;
		panelInput.rightSweeperUpAndInFlag:=FALSE;
	END_IF
END_IF
//右扫盘回收
rTrigger10(CLK:=panelInput.rightSweeperUpAndIn);
IF rTrigger10.Q  THEN
	IF NOT systemStatus.systemWork THEN
		panelInput.rightSweeperOutAndDownFlag:=FALSE;
		panelInput.rightSweeperUpAndInFlag:=TRUE;
	END_IF
END_IF 

//右扫即时摆出，延时3S回收
tof2(IN:=panelInput.rightSweeperOutAndDownFlag,PT:=T#3S);
systemStatus.rightSweeperSwingOut:=tof2.Q AND (NOT systemStatus.systemWork) OR systemStatus.rightSweeperSwingOut;//保证系统工作的情况下，系统工作动作优先
//右扫延时5S下放，控制下放气阀5S得电后失电（保持下放状态）
ton3(IN:=panelInput.rightSweeperOutAndDownFlag,PT:=T#5S);
ton4(IN:=ton3.Q,PT:=T#5S);
systemStatus.rightSweeperDown:=ton3.Q AND (NOT ton4.Q) AND (NOT systemStatus.systemWork) OR systemStatus.rightSweeperDown;//保证系统工作的情况下，系统工作动作优先

END_PROGRAM

// Device/Application/tipsHandle
PROGRAM tipsHandle
VAR
END_VAR

tipsST.highPressurePumpDisconnect:=tipsST.highPressurePumpDisconnect1 OR tipsST.highPressurePumpDisconnect2 OR tipsST.highPressurePumpDisconnect3;//高压水泵未啮合
//tipsST.mainWateraValveNotOpen:=tipsST.mainWateraValveNotOpen1 OR tipsST.mainWateraValveNotOpen2 OR tipsST.mainWateraValveNotOpen3 OR tipsST.mainWateraValveNotOpen4;//总水阀未打开
tipsST.mainWateraValveNotOpen:=tipsST.mainWateraValveNotOpen4;//总水阀未打开
//tipsST.cleanValveNotClose:= tipsST.mainWateraValveNotOpen1 OR tipsST.mainWateraValveNotOpen2 OR tipsST.mainWateraValveNotOpen3 OR tipsST.mainWateraValveNotOpen4;//吹净球阀未打开
tipsST.cleanValveNotClose:= tipsST.mainWateraValveNotOpen4;//吹净球阀未打开

END_PROGRAM

// Device/Application/handleOutput40A
PROGRAM handleOutput40A
VAR
END_VAR

    output40A.connectWaterValve:= ctlTestFlag.ctlConnectWaterValveTest; //连通水阀关闭
	output40A.closeFrontTank:=ctlTestFlag.ctlCloseFrontTankTest; //前水箱关闭
	output40A.cLoseBackTank:=ctlTestFlag.ctlCLoseBackTankTest; //后水箱关闭
	output40A.engineStart:=systemStatus.engineStart; //发动机启动
	output40A.diaphragmPumpStart:=ctlTestFlag.ctlDiaphragmPumpStartTest OR systemStatus.diaphragmPump; //喷雾降尘泵启动
	output40A.backup01:=FALSE; //备用
	output40A.engineStop:=systemStatus.keyRunPosition; //发动机停止
	output40A.sweeperLowSpeed:=ctlTestFlag.ctlSweeperSpeedLowTest OR systemStatus.sweeperSpeedLow; //扫盘低速
	output40A.sweeperMiddleSpeed:=ctlTestFlag.ctlSweeperSpeedMiddleTest OR systemStatus.sweeperSpeedMiddle; //扫盘中速
	output40A.leftAllSweep:=ctlTestFlag.ctlLeftSweeperRotateTest OR systemStatus.leftSweeperRotate OR ctlTestFlag.ctlAllSweeperRotateTest OR systemStatus.allSweeperRotate; //左/全扫
	output40A.rightSweep:=ctlTestFlag.ctlRightSweeperRotateTest OR systemStatus.rightSweeperRotate; //右扫
	output40A.rightAllSweep:=ctlTestFlag.ctlRightSweeperRotateTest OR systemStatus.rightSweeperRotate OR ctlTestFlag.ctlAllSweeperRotateTest OR systemStatus.allSweeperRotate; //右/全扫
	output40A.tankDown:=ctlTestFlag.ctlTankDownTest OR systemStatus.tankDown OR panelInput.tankDownFlag; //箱体降
	output40A.tankUp:=ctlTestFlag.ctlTankUpTest OR systemStatus.tankUp OR panelInput.tankUpFlag; //箱体升
	output40A.suctionNozzleUp:=ctlTestFlag.ctlSuctionNozzleUpTest OR systemStatus.suctionNozzleUp OR panelInput.suctionNozzleUpFlag; //吸嘴升
	output40A.leftBackSprinkle:= ctlTestFlag.ctlLeftBackSprinkleTest OR systemStatus.leftBackSprinkle; //左后洒
	output40A.rightBackSprinkle:= ctlTestFlag.ctlRightBackSprinkleTest OR systemStatus.rightBackSprinkle; //右后洒
	output40A.tankDoorOpen:=ctlTestFlag.ctlTankDoorOpenTest OR systemStatus.tankDoorOpen OR panelInput.tankDoorOpenFlag; //箱门开
	output40A.waterPumpConnect :=ctlTestFlag.ctlWaterPumpConnectTest OR systemStatus.waterPumpConnect; //水泵啮合
	output40A.leftFrontSprinkle:=ctlTestFlag.ctlLeftFrontSprinkleTest OR systemStatus.leftFrontSprinkle; //左前冲
	output40A.rightFrontSprinkle:=ctlTestFlag.ctlRightFrontSprinkleTest OR systemStatus.rightFrontSprinkle; //右前冲
	output40A.suctionNozzleDown:=ctlTestFlag.ctlSuctionNozzleDownTest OR systemStatus.suctionNozzleDown or panelInput.suctionNozzleDownFlag; //吸嘴降
	output40A.tankDoorClose:=ctlTestFlag.ctlTankDoorCloseTest OR systemStatus.tankDoorClose OR panelInput.tankDoorCloseFlag; //箱门关
	output40A.oilUnloadValve:=output40A.tankDown OR output40A.tankUp OR output40A.tankDoorOpen OR output40A.tankDoorClose
      OR output40A.suctionNozzleUp OR output40A.suctionNozzleDown OR  output40A.leftAllSweep OR output40A.rightSweep OR output40A.rightAllSweep; //油路卸荷阀
	
	doConnectWaterValve:=output40A.connectWaterValve; //连通水阀关闭
	doCloseFrontTank:=  output40A.closeFrontTank; //前水箱关闭
	doCLoseBackTank:= output40A.cLoseBackTank; //后水箱关闭
	doEngineStart:= output40A.engineStart; //发动机启动
	doDiaphragmPumpStart:= output40A.diaphragmPumpStart; //隔膜泵启动
	doBackup01:= output40A.backup01; //备用
	doEngineStop:=output40A.engineStop; //发动机停止
	doSweeperLowSpeed:= output40A.sweeperLowSpeed; //扫盘低速
	doSweeperMiddleSpeed:= output40A.sweeperMiddleSpeed; //扫盘中速
	doOilUnloadValve:= output40A.oilUnloadValve; //油路卸荷阀
	doLeftAllSweep:= output40A.leftAllSweep; //左/全扫
	doRightSweep:= output40A.rightSweep; //右扫
	doRightAllSweep:= output40A.rightAllSweep; //右/全扫
	doTankDown:= output40A.tankDown; //箱体降
	doTankUp:= output40A.tankUp; //箱体升
	doSuctionNozzleUp:= output40A.suctionNozzleUp; //吸嘴升
	doLeftBackSprinkle:= output40A.leftBackSprinkle; //左后洒
	doRightBackSprinkle:= output40A.rightBackSprinkle; //右后洒
	doTankDoorOpen:= output40A.tankDoorOpen; //箱门开
	doWaterPumpConnect:= output40A.waterPumpConnect; //水泵啮合
	doLeftFrontSprinkle:= output40A.leftFrontSprinkle; //左前冲
	doRightFrontSprinkle:= output40A.rightFrontSprinkle; //右前冲
	doSuctionNozzleDown:= output40A.suctionNozzleDown; //吸嘴降
	doTankDoorClose:= output40A.tankDoorClose; //箱门关

END_PROGRAM

// Device/Application/handleOutput24B
PROGRAM handleOutput24B
VAR
END_VAR

 
	output24B.auxiliaryValveOpen:= ctlTestFlag.ctlAuxiliaryValueTest OR systemStatus.auxiliaryValveOpen1 OR systemStatus.auxiliaryValveOpen2; //辅助球阀喷水
	output24B.leftSprayRodOpen:= ctlTestFlag.ctlLeftSprayRodOpenTest OR systemStatus.leftSprayRodOpen1 OR systemStatus.leftSprayRodOpen2; //左侧喷杆喷水
	output24B.selfSprayRodOpen:= ctlTestFlag.ctlSelfCleanTest OR systemStatus.selfSprayRodOpen1 OR systemStatus.selfSprayRodOpen2; //自洁喷杆喷水
	output24B.rightSprayRodOpen:= ctlTestFlag.ctlRightSprayRodOpenTest OR systemStatus.rightSprayRodOpen1 OR  systemStatus.rightSprayRodOpen2; //右侧喷杆喷水
	output24B.centreSprayRodOpen:= ctlTestFlag.ctlCentreSprayRodOpenTest OR systemStatus.centreSprayRodOpen1 OR systemStatus.centreSprayRodOpen2 ; //中喷杆喷水
	output24B.waterUnloadValveOpen:=output24B.auxiliaryValveOpen OR output24B.leftSprayRodOpen OR output24B.selfSprayRodOpen
    OR output24B.rightSprayRodOpen OR output24B.centreSprayRodOpen ; //卸荷球阀打开
	
	output24B.engineDisconect:=  ctlTestFlag.ctlEngineDisconnectTest OR systemStatus.engineDisconect;  //副发分离
	output24B.backupEngineStart:= systemStatus.backupMotorOpen; //备用动力
	output24B.rightSweeperDown:= ctlTestFlag.ctlRightSweeperDownTest OR systemStatus.rightSweeperDown; //右扫降
	output24B.rightSweeperUp:= ctlTestFlag.ctlRightSweeperUpTest OR systemStatus.rightSweeperUp; //右扫升
	output24B.leftSweeperSwingOut :=ctlTestFlag.ctlLeftSweeperSwingOutTest OR systemStatus.leftSweeperSwingOut; //左扫摆出
	output24B.rightSweeperSwingOut:= ctlTestFlag.ctlRightSweeperSwingOutTest OR systemStatus.rightSweeperSwingOut; //右扫摆出
	output24B.leftSprayRodSwingOut := ctlTestFlag.ctlLeftSprayRodSwingOutTest OR systemStatus.leftSprayRodSwingOut OR panelInput.sprayRodOutOrInFlag; //左侧喷杆摆出
	output24B.rightSprayRodSwingOut:= ctlTestFlag.ctlRightSprayRodSwingOutTest OR systemStatus.rightSprayRodSwingOut OR panelInput.sprayRodOutOrInFlag; //右侧喷杆摆出
	output24B.leftSweeperDown:= ctlTestFlag.ctlLeftSweeperDownTest OR systemStatus.leftSweeperDown; //左扫盘降
	output24B.leftSweeperUp:= ctlTestFlag.ctlLeftSweeperUpTest OR systemStatus.leftSweeperUp;  //左扫盘升
	
	doWaterUnloadValveOpen:= output24B.waterUnloadValveOpen; //卸荷球阀打开
	doAuxiliaryValveOpen:= output24B.auxiliaryValveOpen; //辅助球阀喷水
	doLeftSprayRodOpen := output24B.leftSprayRodOpen; //左侧喷杆喷水
	doSelfSprayRodOpen := output24B.selfSprayRodOpen; //自洁喷杆喷水
	doRightSprayRodOpen := output24B.rightSprayRodOpen; //右侧喷杆喷水
	doCentreSprayRodOpen:= output24B.centreSprayRodOpen; //中喷杆喷水
	doEngineDisconect:= output24B.engineDisconect;  //副发分离
	doBackupEngineStart:=  output24B.backupEngineStart; //备用动力
	doRightSweeperDown:= output24B.rightSweeperDown; //右扫降
	doRightSweeperUp := output24B.rightSweeperUp; //右扫升
	doLeftSweeperSwingOut:= output24B.leftSweeperSwingOut; //左扫摆出
	doRightSweeperSwingOut:= output24B.rightSweeperSwingOut; //右扫摆出
	doLeftSprayRodSwingOut:=  output24B.leftSprayRodSwingOut; //左侧喷杆摆出
	doRightSprayRodSwingOut:= output24B.rightSprayRodSwingOut ; //右侧喷杆摆出
	doLeftSweeperDown :=output24B.leftSweeperDown; //左扫盘降
	doLeftSweeperUp:= output24B.leftSweeperUp;  //左扫盘升

END_PROGRAM

// Device/Application/transmit2HMI
PROGRAM transmit2HMI
VAR
	sndCAN: JCMC_Ctrl.CAN_TRANSMIT;//can发送
	sendBuf1:JCMC_Ctrl.CanMsgST;//控制器发送给触摸屏报文包1,CAN1,0x18004F2A
	sendBuf2:JCMC_Ctrl.CanMsgST;//控制器发送给触摸屏报文包2,CAN1,0x18014F2A
	sendBuf3:JCMC_Ctrl.CanMsgST;//控制器发送给触摸屏报文包3,CAN1,0x18024F2A
	sendBuf4:JCMC_Ctrl.CanMsgST;//控制器发送给触摸屏报文包4,CAN1,0x18034F2A
	sendBuf5:JCMC_Ctrl.CanMsgST;//控制器发送给触摸屏报文包5,CAN1,0x18044F2A
	sendBuf6:JCMC_Ctrl.CanMsgST;//控制器发送给触摸屏报文包6,CAN1,0x18054F2A
	
	ton1:TON;//0x18004F2A,发送周期100ms
	ton2:TON;//0x18014F2A,发送周期100ms
	ton3:TON;//0x18024F2A,发送周期100ms
	ton4:TON;//0x18034F2A,发送周期100ms
	ton5:TON;//0x18044F2A,发送周期100ms
	ton6:TON;//0x18054F2A,发送周期100ms
END_VAR

//控制器发送给触摸屏报文包1,0x18004F2A
sendBuf1.Data[0].1:=faultSt.coolingTankWaterLevelLow;//冷却水箱液位低
sendBuf1.Data[0].2:=input24B.generatorWork; //发电机发电
sendBuf1.Data[0].5:=input24B.waitingStartLamp; //等待启动灯
sendBuf1.Data[0].6:=input24B.alarmLamp; //警告故障灯
sendBuf1.Data[0].7:=input24B.stopEngineLamp; //停机故障灯

sendBuf1.Data[1].0:=input40A.diaphragmPumpPressure; //隔膜泵压力正常
sendBuf1.Data[1].1:=input40A.mainWateraValve;//总水阀接近开关
sendBuf1.Data[1].2:=input40A.cleanValve;//吹净球阀接近开关
sendBuf1.Data[1].3:=input40A.backDoor;//后门接近开关
sendBuf1.Data[1].4:=input40A.waterUnloadValve;//水路卸荷阀接近开关
sendBuf1.Data[1].5:=input40A.leftRod;//左侧撑杆接近开关
sendBuf1.Data[1].6:=input40A.rightRod;//右侧撑杆接近开关
sendBuf1.Data[1].7:=input24B.reverseCar;//倒车

sendBuf1.Data[3].0:=faultST.alarmLamp;//发动机警告故障
sendBuf1.Data[3].1:=faultST.stopEngineLamp;   //发动机停机故障
sendBuf1.Data[3].2:=faultST.coolingTankWaterLevelLow;//冷却水箱液位低
sendBuf1.Data[3].3:=faultST.waterUnloadValveNotClose;	//水路卸荷阀未关闭
sendBuf1.Data[3].4:=faultST.waterUnloadValveNotOpen;	//水路卸荷阀未打开
sendBuf1.Data[3].5:=faultST.bilgeTankFull;	//污水满
sendBuf1.Data[3].6:=faultST.returnOilFilterBlockUp;	//回油过滤堵塞
sendBuf1.Data[3].7:=faultST.hHighPressureFilterBlockUp;	//高压油滤堵塞

sendBuf1.Data[4].0:=faultST.hydraulicOilLevelLow;	//液压油位低
sendBuf1.Data[4].1:=faultST.frontTankWaterLevelLow;	//前水箱缺水
sendBuf1.Data[4].2:=faultST.backTankWaterLevelLow;	//后水箱缺水
sendBuf1.Data[4].3:=faultST.tankWaterLevelLow;	//水箱缺水
sendBuf1.Data[4].4:=faultST.reverseCarStop;	//倒车故障停机
sendBuf1.Data[4].5:=faultST.waterFullStop;	//污水满故障停机
sendBuf1.Data[4].6:=faultST.highPressurePumpOverSpeedAlarm;	//高压水泵超速报警
sendBuf1.Data[4].7:=faultST.highPressurePumpOverSpeedStop;	//高压水泵超速停止

sendBuf1.Data[5].0:=faultST.diaphragmPumpPressure;	//喷雾降尘泵故障
sendBuf1.Data[5].1:=tipsST.closeTest;	//请关闭测试
sendBuf1.Data[5].2:=tipsST.reverseCar;	//正在倒车中
sendBuf1.Data[5].3:=tipsST.startEngineFirst;	//请先打开发动机
sendBuf1.Data[5].4:=tipsST.backupMotorOpen;	//备用动力打开
sendBuf1.Data[5].5:=tipsST.testOpen;	//测试打开
sendBuf1.Data[5].6:=tipsST.highPressurePumpDisconnect;	//高压水泵未啮合
sendBuf1.Data[5].7:=tipsST.tankDoorNotOpen; //箱门未打开

sendBuf1.Data[6].1:=tipsST.leftRodUp;	//左支撑杆未放下
sendBuf1.Data[6].2:=tipsST.rightRodUp;	//右支撑杆未放下
sendBuf1.Data[6].3:=tipsST.mainWateraValveNotOpen;	//总水阀未打开
sendBuf1.Data[6].4:=tipsST.cleanValveNotClose;	//吹净球阀未关闭

sendBuf1.ID:=16#18004F2A;
ton1(IN:=NOT ton1.Q ,PT:=T#100MS);
IF ton1.Q THEN
	sndCAN(CHANNEL:=1,ENABLE:=TRUE,ID:=sendBuf1.ID,DLC:=8,DATA:=sendBuf1.Data);
	IF NOT sndCAN.RESULT THEN
	//do nothing
	END_IF
END_IF


//控制器发送给触摸屏报文包2,CAN1,0x18014F2A
//发动机工作小时
sendBuf2.Data[3]:=WORD_TO_BYTE(DWORD_TO_WORD(SHR(systemStatus.engineWorkTime,16)/256));
sendBuf2.Data[2]:=WORD_TO_BYTE(DWORD_TO_WORD(SHR(systemStatus.engineWorkTime,16)));
sendBuf2.Data[1]:=WORD_TO_BYTE(DWORD_TO_WORD(systemStatus.engineWorkTime)/256);
sendBuf2.Data[0]:=WORD_TO_BYTE(DWORD_TO_WORD(systemStatus.engineWorkTime));
//副发转速
sendBuf2.Data[4]:=WORD_TO_BYTE(systemStatus.engineRealSpeed);
sendBuf2.Data[5]:=WORD_TO_BYTE(systemStatus.engineRealSpeed/256);
//副发水温
sendBuf2.Data[6]:=SINT_TO_BYTE(systemStatus.engineCoolingTemperature+40);
//副发油压
sendBuf2.Data[7]:=systemStatus.engineOilPressure/4;

sendBuf2.ID:=16#18014F2A;
ton2(IN:=NOT ton2.Q ,PT:=T#100MS);
IF ton2.Q THEN
	sndCAN(CHANNEL:=1,ENABLE:=TRUE,ID:=sendBuf2.ID,DLC:=8,DATA:=sendBuf2.Data);
	IF NOT sndCAN.RESULT THEN
	//do nothing
	END_IF
END_IF

//控制器发送给触摸屏报文包3,CAN1,0x18024F2A
//系统剩余工作时间
sendBuf3.Data[0]:=WORD_TO_BYTE(systemStatus.systemEndurance);
sendBuf3.Data[1]:=WORD_TO_BYTE(systemStatus.systemEndurance/256);
//剩余水量
sendBuf3.Data[2]:=WORD_TO_BYTE(100*systemStatus.systemEndurance);
sendBuf3.Data[3]:=WORD_TO_BYTE(100*systemStatus.systemEndurance/256);
//控制器版本
sendBuf3.Data[4]:=WORD_TO_BYTE(systemStatus.softVersion);
sendBuf3.Data[5]:=WORD_TO_BYTE(systemStatus.softVersion/256);

sendBuf3.ID:=16#18034F2A;
ton3(IN:=NOT ton3.Q ,PT:=T#100MS);
IF ton3.Q THEN
	sndCAN(CHANNEL:=1,ENABLE:=TRUE,ID:=sendBuf3.ID,DLC:=8,DATA:=sendBuf3.Data);
	IF NOT sndCAN.RESULT THEN
		//do nothing
	END_IF
END_IF

//控制器发送给触摸屏报文包4,CAN1,0x18034F2A
//垃圾箱负压
sendBuf4.Data[0]:=WORD_TO_BYTE(input40A.dumpsterPressure);
sendBuf4.Data[1]:=WORD_TO_BYTE(input40A.dumpsterPressure/256);
//吸桶负压
sendBuf4.Data[2]:=WORD_TO_BYTE(input40A.suctionBucketPressure);
sendBuf4.Data[3]:=WORD_TO_BYTE(input40A.suctionBucketPressure/256);
//前水箱水位
sendBuf4.Data[4]:=WORD_TO_BYTE(input40A.frontWaterTankPressure);
sendBuf4.Data[5]:=WORD_TO_BYTE(input40A.frontWaterTankPressure/256);
//后水箱水位
sendBuf4.Data[6]:=WORD_TO_BYTE(input40A.backWaterTankPressure);
sendBuf4.Data[7]:=WORD_TO_BYTE(input40A.backWaterTankPressure/256);

sendBuf4.ID:=16#18034F2A;
ton4(IN:=NOT ton4.Q ,PT:=T#100MS);
IF ton4.Q THEN
	sndCAN(CHANNEL:=1,ENABLE:=TRUE,ID:=sendBuf4.ID,DLC:=8,DATA:=sendBuf4.Data);
	IF NOT sndCAN.RESULT THEN
		//do nothing
	END_IF
END_IF

//控制器发送给触摸屏报文包5,CAN1,0x18044F2A
sendBuf5.Data[0].0:=output40A.connectWaterValve; //连通水阀关闭
sendBuf5.Data[0].1:=output40A.closeFrontTank; //前水箱关闭
sendBuf5.Data[0].2:=output40A.cLoseBackTank; //后水箱关闭
sendBuf5.Data[0].3:=output40A.engineStart; //发动机启动
sendBuf5.Data[0].4:=output40A.diaphragmPumpStart; //喷雾降尘泵启动
sendBuf5.Data[0].5:=output40A.backup01; //备用
sendBuf5.Data[0].6:=output40A.engineStop; //发动机停止
sendBuf5.Data[0].7:=output40A.sweeperLowSpeed; //扫盘低速

sendBuf5.Data[1].0:=output40A.sweeperMiddleSpeed; //扫盘中速
sendBuf5.Data[1].1:=output40A.oilUnloadValve; //油路卸荷阀
sendBuf5.Data[1].2:=output40A.leftAllSweep; //左/全扫
sendBuf5.Data[1].3:=output40A.rightSweep; //右扫
sendBuf5.Data[1].4:=output40A.rightAllSweep; //右/全扫
sendBuf5.Data[1].5:=output40A.tankDown; //箱体降
sendBuf5.Data[1].6:=output40A.tankUp; //箱体升
sendBuf5.Data[1].7:=output40A.suctionNozzleUp; //吸嘴升

sendBuf5.Data[2].0:=output40A.leftBackSprinkle; //左后洒
sendBuf5.Data[2].1:=output40A.rightBackSprinkle; //右后洒
sendBuf5.Data[2].2:=output40A.tankDoorOpen; //箱门开
sendBuf5.Data[2].3:=output40A.waterPumpConnect; //水泵啮合
sendBuf5.Data[2].4:=output40A.leftFrontSprinkle; //左前冲
sendBuf5.Data[2].5:=output40A.rightFrontSprinkle; //右前冲
sendBuf5.Data[2].6:=output40A.suctionNozzleDown; //吸嘴降
sendBuf5.Data[2].7:=output40A.tankDoorClose; //箱门关

sendBuf5.Data[3].0:=output24B.waterUnloadValveOpen; //卸荷球阀打开
sendBuf5.Data[3].1:=output24B.auxiliaryValveOpen; //辅助球阀喷水
sendBuf5.Data[3].2:=output24B.leftSprayRodOpen; //左侧喷杆喷水
sendBuf5.Data[3].3:=output24B.selfSprayRodOpen; //自洁喷杆喷水
sendBuf5.Data[3].4:=output24B.rightSprayRodOpen; //右侧喷杆喷水
sendBuf5.Data[3].5:=output24B.centreSprayRodOpen; //中喷杆喷水
sendBuf5.Data[3].6:=output24B.engineDisconect;  //副发分离
sendBuf5.Data[3].7:=output24B.backupEngineStart; //备用动力

sendBuf5.Data[4].0:=output24B.rightSweeperDown; //右扫降
sendBuf5.Data[4].1:=output24B.rightSweeperUp; //右扫升
sendBuf5.Data[4].2:=output24B.leftSweeperSwingOut; //左扫摆出
sendBuf5.Data[4].3:=output24B.rightSweeperSwingOut; //右扫摆出
sendBuf5.Data[4].4:=output24B.leftSprayRodSwingOut; //左侧喷杆摆出
sendBuf5.Data[4].5:=output24B.rightSprayRodSwingOut; //右侧喷杆摆出
sendBuf5.Data[4].6:=output24B.leftSweeperDown; //左扫盘降
sendBuf5.Data[4].7:=output24B.leftSweeperUp;  //左扫盘升
	
sendBuf5.ID:=16#18044F2A;
ton5(IN:=NOT ton5.Q ,PT:=T#100MS);
IF ton5.Q THEN
	sndCAN(CHANNEL:=1,ENABLE:=TRUE,ID:=sendBuf5.ID,DLC:=8,DATA:=sendBuf5.Data);
	IF NOT sndCAN.RESULT THEN
		//do nothing
	END_IF
END_IF

//控制器发送给触摸屏报文包6,CAN1,0x18054F2A
sendBuf6.Data[0].0:=systemStatus.systemWork;//系统工作状态
sendBuf6.Data[0].1:=systemStatus.keyRunPosition; //钥匙运行档标志
sendBuf6.Data[0].2:=systemStatus.engineStart; //发动机启动标志
sendBuf6.Data[0].3:=systemStatus.standardSpeed;	//标准速度标志
sendBuf6.Data[0].4:=systemStatus.strongSpeed;	//强力速度标志
sendBuf6.Data[0].5:=systemStatus.allWashSweep;	//全洗扫状态
sendBuf6.Data[0].6:=systemStatus.leftWashSweep;	//左洗扫状态
sendBuf6.Data[0].7:=systemStatus.rightWashSweep;	//右洗扫状态

sendBuf6.Data[1].0:=systemStatus.allSweep;	//全扫路状态
sendBuf6.Data[1].1:=systemStatus.leftSweep;	//左扫路状态
sendBuf6.Data[1].2:=systemStatus.rightSweep;	//右扫路状态
sendBuf6.Data[1].3:=systemStatus.allWash;	//全清洗状态
sendBuf6.Data[1].4:=systemStatus.leftWash;	//左清洗状态
sendBuf6.Data[1].5:=systemStatus.rightWash;	//右清洗状态
sendBuf6.Data[1].6:=systemStatus.stopWash;	//停扫状态
sendBuf6.Data[1].7:=systemStatus.leftFlushOpen;	//左角冲打开标志

sendBuf6.Data[2].0:=systemStatus.rightFlushOpen;	//右角冲打开标志
sendBuf6.Data[2].1:=systemStatus.backSprayOpen;	//后喷雾打开标志
sendBuf6.Data[2].2:=systemStatus.sprayGun;	//手持喷枪打开标志
sendBuf6.Data[2].3:=systemStatus.selfClean;	//	自洁打开标志
sendBuf6.Data[2].4:=systemStatus.leftFrontSprinkle;	//	左前冲打开标志
sendBuf6.Data[2].5:=systemStatus.rightFrontSprinkle;	//	右前冲打开标志
sendBuf6.Data[2].6:=systemStatus.leftBackSprinkle;	//	左后洒打开标志
sendBuf6.Data[2].7:=systemStatus.rightBackSprinkle;	//	右后洒打开标志

sendBuf6.Data[3].0:=systemStatus.replaceSweeper;	//更换扫刷标志
sendBuf6.Data[3].6:=ctlTestFlag.ctlLeftBackSprinkleTest;	//	左后洒_测试_控制器
sendBuf6.Data[3].7:=ctlTestFlag.ctlRightBackSprinkleTest;	//	右后洒_测试_控制器

sendBuf6.Data[4].0:=ctlTestFlag.ctlEngineDisconnectTest;	//副发分离_测试_控制器
sendBuf6.Data[4].1:=ctlTestFlag.ctlConnectWaterValveTest;	//连通水阀_测试_控制器
sendBuf6.Data[4].2:=ctlTestFlag.ctlCloseFrontTankTest;	//前水箱水阀_测试_控制器
sendBuf6.Data[4].3:=ctlTestFlag.ctlCLoseBackTankTest;	//后水箱水阀_测试_控制器
sendBuf6.Data[4].4:=ctlTestFlag.ctlSweeperSpeedLowTest;	//扫盘低速_测试_控制器
sendBuf6.Data[4].5:=ctlTestFlag.ctlSweeperSpeedMiddleTest;	//扫盘中速_测试_控制器
sendBuf6.Data[4].6:=ctlTestFlag.ctlLeftSweeperRotateTest;	//左扫旋转_测试_控制器
sendBuf6.Data[4].7:=ctlTestFlag.ctlRightSweeperRotateTest;	//右扫旋转_测试_控制器

sendBuf6.Data[5].0:=ctlTestFlag.ctlAllSweeperRotateTest;	//全扫旋转_测试_控制器
sendBuf6.Data[5].1:=ctlTestFlag.ctlTankDownTest;	//箱体降_测试_控制器
sendBuf6.Data[5].2:=ctlTestFlag.ctlTankUpTest;	//箱体升_测试_控制器
sendBuf6.Data[5].3:=ctlTestFlag.ctlSuctionNozzleDownTest;	//吸嘴降_测试_控制器
sendBuf6.Data[5].4:=ctlTestFlag.ctlSuctionNozzleUpTest;	//吸嘴升_测试_控制器
sendBuf6.Data[5].5:=ctlTestFlag.ctlTankDoorOpenTest;	//箱门开_测试_控制器
sendBuf6.Data[5].6:=ctlTestFlag.ctlTankDoorCloseTest;	//箱门关_测试_控制器
sendBuf6.Data[5].7:=ctlTestFlag.ctlLeftSweeperDownTest;	//左扫盘下放_测试_控制器

sendBuf6.Data[6].0:=ctlTestFlag.ctlLeftSweeperUpTest;	//左扫盘回收_测试_控制器
sendBuf6.Data[6].1:=ctlTestFlag.ctlRightSweeperDownTest;	//右扫盘下放_测试_控制器
sendBuf6.Data[6].2:=ctlTestFlag.ctlRightSweeperUpTest;	//右扫盘回收_测试_控制器
sendBuf6.Data[6].3:=ctlTestFlag.ctlLeftSweeperSwingOutTest;	//左扫盘摆出_测试_控制器
sendBuf6.Data[6].4:=ctlTestFlag.ctlRightSweeperSwingOutTest;	//右扫盘摆出_测试_控制器
sendBuf6.Data[6].5:=ctlTestFlag.ctlLeftSprayRodSwingOutTest;	//左喷杆摆出_测试_控制器
sendBuf6.Data[6].6:=ctlTestFlag.ctlRightSprayRodSwingOutTest;	//右喷杆摆出_测试_控制器
sendBuf6.Data[6].7:=ctlTestFlag.ctlLeftSprayRodOpenTest;	//左喷杆喷水_测试_控制器
    
sendBuf6.Data[7].0:=ctlTestFlag.ctlRightSprayRodOpenTest;	//右喷杆喷水_测试_控制器
sendBuf6.Data[7].1:=ctlTestFlag.ctlCentreSprayRodOpenTest;	//中喷杆喷水_测试_控制器
sendBuf6.Data[7].2:=ctlTestFlag.ctlAuxiliaryValueTest;	//辅助球阀打开_测试_控制器
sendBuf6.Data[7].3:=ctlTestFlag.ctlSelfCleanTest;	//自洁打开_测试_控制器
sendBuf6.Data[7].4:=ctlTestFlag.ctlWaterPumpConnectTest;	//高压水泵啮合_测试_控制器
sendBuf6.Data[7].5:=ctlTestFlag.ctlDiaphragmPumpStartTest;	//喷雾降尘泵_测试_控制器
sendBuf6.Data[7].6:=ctlTestFlag.ctlLeftFrontSprinkleTest;	//	左前冲_测试_控制器
sendBuf6.Data[7].7:=ctlTestFlag.ctlRightFrontSprinkleTest;	//	右前冲_测试_控制器  
    
sendBuf6.ID:=16#18054F2A;
ton6(IN:=NOT ton6.Q ,PT:=T#100MS);
IF ton6.Q THEN
	sndCAN(CHANNEL:=1,ENABLE:=TRUE,ID:=sendBuf6.ID,DLC:=8,DATA:=sendBuf6.Data);
	IF NOT sndCAN.RESULT THEN
		//do nothing
	END_IF   
END_IF

END_PROGRAM

// Device/Application/transmit2SiliconePanel
PROGRAM transmit2SiliconePanel
VAR
	sndCAN: JCMC_Ctrl.CAN_TRANSMIT;//can发送
	sendBuf1:JCMC_Ctrl.CanMsgST;//控制器发送给硅胶面板 报文包1,CAN1,0x0801F02A,100ms循环
	sendBuf2:JCMC_Ctrl.CanMsgST;//控制器发送给硅胶面板 报文包2,CAN1,0x0802F02A,100ms循环
	sendBuf3:JCMC_Ctrl.CanMsgST;//控制器发送给硅胶面板 报文包3,CAN1,0x00000505,按需发送
	
	ton1:TON;//0x0801F02A,发送周期100ms
	ton2:TON;//0x0802F02A,发送周期100ms
	ton3:TON;//0x00000505,发送周期100ms
	rTrigger1:R_TRIG;//工作灯标志上升沿触发
END_VAR

//控制器发送给硅胶面板 报文包1,CAN1,0x0801F02A,100ms循环
sendBuf1.Data[0].2:=panelInput.tankDoorOpenFlag;	//垃圾箱门开_硅胶面板_返回标志
sendBuf1.Data[1].2:=panelInput.tankDoorCloseFlag;	//垃圾箱门关_硅胶面板_返回标志
sendBuf1.Data[2].2:=panelInput.tankUpFlag;	//垃圾箱体升_硅胶面板_返回标志
sendBuf1.Data[3].2:=panelInput.tankDownFlag;	//垃圾箱体降_硅胶面板_返回标志
sendBuf1.Data[4].2:=panelInput.leftSweeperUpAndInFlag;	//左扫盘回收_硅胶面板_返回标志
sendBuf1.Data[5].2:=panelInput.leftSweeperOutAndDownFlag;	//左扫盘下放_硅胶面板_返回标志
sendBuf1.Data[6].2:=panelInput.rightSweeperUpAndInFlag;	//右扫盘回收_硅胶面板_返回标志
sendBuf1.Data[7].2:=panelInput.rightSweeperOutAndDownFlag;	//右扫盘下放_硅胶面板_返回标志

sendBuf1.ID:=16#0801F02A;
ton1(IN:=NOT ton1.Q ,PT:=T#100MS);
IF ton1.Q THEN
	sndCAN(CHANNEL:=1,ENABLE:=TRUE,ID:=sendBuf1.ID,DLC:=8,DATA:=sendBuf1.Data);
	IF NOT sndCAN.RESULT THEN
		//do nothing
	END_IF
END_IF

//控制器发送给硅胶面板 报文包2,CAN1,0x0802F02A,100ms循环
sendBuf2.Data[0].2:=panelInput.suctionNozzleUpFlag;	//吸嘴升_硅胶面板_返回标志
sendBuf2.Data[1].2:=panelInput.suctionNozzleDownFlag;	//吸嘴降_测试_硅胶面板_返回标志
sendBuf2.Data[2].2:=panelInput.selfCleanFlag;	//自洁打开_硅胶面板_返回标志
sendBuf2.Data[3].2:=panelInput.sprayGunFlag;	//手持喷枪_硅胶面板_返回标志
sendBuf2.Data[4].2:=panelInput.sprayRodOutOrInFlag;  //喷杆伸缩_硅胶面板_返回标志
sendBuf2.Data[5].2:=panelInput.backupMotorFlag; //备用动力_硅胶面板_返回标志
sendBuf2.Data[6].2:=panelInput.workLampFlag; //工作灯_硅胶面板_返回标志
sendBuf2.Data[7].2:=panelInput.backlightFlag; //背光灯_硅胶面板_返回标志

sendBuf1.ID:=16#0802F02A;
ton2(IN:=NOT ton2.Q ,PT:=T#100MS);
IF ton2.Q THEN
	sndCAN(CHANNEL:=1,ENABLE:=TRUE,ID:=sendBuf1.ID,DLC:=8,DATA:=sendBuf2.Data);
	IF NOT sndCAN.RESULT THEN
		//do nothing
	END_IF
END_IF

//控制器发送给硅胶面板 报文包3,CAN1,0x00000505,按需发送
sendBuf3.Data[0].0:=1;//扩展帧
sendBuf3.Data[0].1:=panelInput.backlightFlag;//背光开关
sendBuf3.Data[0].2:=1;//输出控制、
sendBuf3.Data[0].3:=0;//无定义
sendBuf3.Data[0].4:=0;//0：不动作，1：重启动
sendBuf3.Data[0].5:=0;//无定义
sendBuf3.Data[0].6:=0;//无定义
sendBuf3.Data[0].7:=0;//无定义
sendBuf3.Data[1]:=16#0A;//按键发送周期100ms
sendBuf3.Data[2]:=16#0A;//LED灯接收周期
sendBuf3.Data[3]:=16#00;//CAN波特率
sendBuf3.Data[4]:=16#64;//指示灯亮度
sendBuf3.Data[5]:=16#00;//保留
sendBuf3.Data[6]:=16#00;//保留
sendBuf3.Data[7]:=16#00;//保留

sendBuf1.ID:=16#00000505;
rTrigger1(clk:=panelInput.workLampFlag);
IF   rTrigger1.Q   THEN 
	sndCAN(CHANNEL:=1,ENABLE:=TRUE,ID:=sendBuf3.ID,DLC:=8,DATA:=sendBuf3.Data);
	IF NOT sndCAN.RESULT THEN
		//do nothing
	END_IF
END_IF

END_PROGRAM

// Device/Application/transmit2EngineECM
PROGRAM transmit2EngineECM
VAR
	sndCAN: JCMC_Ctrl.CAN_TRANSMIT;//can发送
	sendBuf1:JCMC_Ctrl.CanMsgST;//控制器发送给副发动机 报文包1,CAN1,0x18EA0007,每秒1次
	sendBuf2:JCMC_Ctrl.CanMsgST;//控制器发送给副发动机 报文包2,CAN1,0x0C000007,10ms循环
	ton1:ton;//发送给副发请求定时器
END_VAR

//控制器发送给副发动机 报文包1,CAN1,0x18EA0007,每秒1次
//请求发动机运行时间 PGN=65253（0xFEE5）
sendBuf1.Data[0]:=16#E5;
sendBuf1.Data[1]:=16#FE;
sendBuf1.Data[2]:=16#00;
sendBuf1.Data[3]:=16#FF;
sendBuf1.Data[4]:=16#FF;
sendBuf1.Data[5]:=16#FF;
sendBuf1.Data[6]:=16#FF;
sendBuf1.Data[7]:=16#FF;

sendBuf1.ID:=16#18EA0007;
ton1(IN:=(NOT ton1.Q),PT:=T#1S);
IF ton1.Q THEN 
	sndCAN(CHANNEL:=1,ENABLE:=TRUE,ID:=sendBuf1.ID,DLC:=8,DATA:=sendBuf1.Data);
	IF NOT sndCAN.RESULT THEN
		//do nothing
	END_IF
END_IF

//控制器发送给副发动机 报文包2,CAN1,0x0C000007,10ms循环
sendBuf2.Data[0]:=16#F5;//速度控制模式
sendBuf2.Data[1]:=WORD_TO_BYTE(8*systemStatus.engineSetSpeed);//给定速度
sendBuf2.Data[2]:=WORD_TO_BYTE(8*systemStatus.engineSetSpeed/256);//给定速度
sendBuf2.Data[3]:=16#FF;//
sendBuf2.Data[4]:=16#FF;
sendBuf2.Data[5]:=16#FF;
sendBuf2.Data[6]:=16#FF;
sendBuf2.Data[7]:=16#FF;

sndCAN(CHANNEL:=1,ENABLE:=TRUE,ID:=sendBuf2.ID,DLC:=8,DATA:=sendBuf2.Data);
IF NOT sndCAN.RESULT THEN
	//do nothing
END_IF

END_PROGRAM

// Device/Application/receiveFromVoiceAlarm
PROGRAM receiveFromVoiceAlarm
VAR
END_VAR

END_PROGRAM
